{attribute 'GeneratedUsingTerminal: EK1100-0000-0018'}
{attribute addProperty BoxType "EK1100-0000-0018"}
{attribute addProperty Id "Beckhoff_EPP2xxxEK1122Beckhoff_EPP2xxxEK1122_76AF9B9A2100"}
{attribute addProperty CRC "282674543"}
{attribute addProperty Size "2100"}
TYPE Beckhoff_EPP2xxx_10D9456F EXTENDS EK1100_AB5A9467 :
STRUCT
	{attribute addProperty Name "Beckhoff_EPP2xxxEK1122"}
	{attribute addProperty PreviousPort "Beckhoff EPP2xxx : B"}
	Beckhoff_EPP2xxxEK1122 : Beckhoff_EPP2xxxEK1122_76AF9B9A;
END_STRUCT
END_TYPE

(* stored: Version 1.2.0.0, ProductVersion 3.1.4024.9
   DUT Beckhoff_EPP2xxx_10D9456F: Id {f44aac93-c6ad-469c-821f-664162139036} *)
